// TIA Portal V20 export
DATA_BLOCK "DB_Digital_Input"   // DB1
{ S7_Optimized_Access := 'TRUE' }
// stored: MemoryReserve 100
   VAR
      Emergency_Stop_Release : Bool;
      Sensor_Water_Fountain_Before_Entrace_Functional_Test_Spinner_Conveyor_Belt : Bool;
      Sensor_Water_Fountain_Entrace_Functional_Test_Spinner_Conveyor_Belt : Bool;
      Sensor_Water_Fountain_Entrace_Functional_Test_After_Spinner_Conveyor_Belt : Bool;
      Trigger_Read_Serial_Number_Entrace_Functional_Test : Bool;
      Sensor_Water_Fountain_Geting_Exit_Rework_Conveyor_Belt : Bool;
      Button_Water_Fountain_Get_Exit_Rework_Conveyor_Belt : Bool;
      Trigger_Read_Serial_Number_Exit_Functional_Test : Bool;
      Sensor_Water_Fountain_Exit_Functional_Test_Spinner_Conveyor_Belt : Bool;
      Sensor_Water_Fountain_Exit_Functional_Test_After_Spinner_Conveyor_Belt : Bool;
      Sensor_Water_Fountain_Geting_Entrace_Rework_Conveyor_Belt_Start : Bool;
      Sensor_Water_Fountain_Geting_Entrace_Rework_Conveyor_Belt_Finish : Bool;
      Carousel_Frequency_Inverter_Fail : Bool;
      Conveyor_Belt_Functional_Test_Inverter_Fail : Bool;
      Selected_Voltage_220V : Bool;
      Selected_Voltage_127V : Bool;
      Sensor_Spinner_Entrace_Functional_Test_Position_Withdrawn : Bool;
      Sensor_Spinner_Entrace_Functional_Test_Position_Advanced : Bool;
      Sensor_Spinner_Exit_Functional_Test_Position_Withdrawn : Bool;
      Sensor_Spinner_Exit_Functional_Test_Position_Advanced : Bool;
      Digital_Input_20 : Bool;
      Digital_Input_21 : Bool;
      Digital_Input_22 : Bool;
      Digital_Input_23 : Bool;
      Digital_Input_24 : Bool;
      Digital_Input_25 : Bool;
      Digital_Input_26 : Bool;
      Digital_Input_27 : Bool;
      Digital_Input_28 : Bool;
      Digital_Input_29 : Bool;
   END_VAR
BEGIN
END_DATA_BLOCK
